TYPE TcoUrRobotics_Config_v_1_x_x :
STRUCT
    InfoTime : TIME := T#2S;
    ErrorTime : TIME := T#0S;
    RemotePowerOnEnabled : BOOL := FALSE;
    RemotePowerOnPulse : TIME := T#500MS;
    IpAddress : STRING;
END_STRUCT
END_TYPE

(* stored: Version 1.1.0.1, ProductVersion 3.1.4024.12
   DUT TcoUrRobotics_Config_v_1_x_x: Id {29ee9b4f-6cb9-0066-239b-3bf709e7eeb1} *)
